% RSLogix 500 project SARUUU_BAK000.RSS, saved by version 8.10.00.18 %
PROJECT "UNTITLED"    % processor: MicroLogix 1200 %

PROGRAM FILES
  LAD 2   3 rungs

DATA FILES
  O0 OUTPUT  4 elements
  I1 INPUT  4 elements
  S2 STATUS  66 elements
  B3 BINARY  1 elements
  T4 TIMER  1 elements
  C5 COUNTER  1 elements
  R6 CONTROL  1 elements
  N7 INTEGER  1 elements

LADDER 2
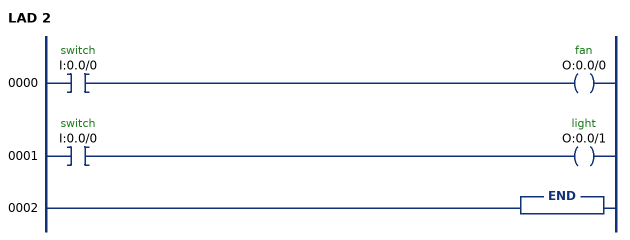
% Rung: 0 %  % edit flag set %
SOR XIC I:0.0/0 OTE O:0.0/0 EOR
%   I:0.0/0  "switch" %
%   O:0.0/0  "fan" %
% Rung: 1 %  % edit flag set %
SOR XIC I:0.0/0 OTE O:0.0/1 EOR
%   I:0.0/0  "switch" %
%   O:0.0/1  "light" %
% Rung: 2 %
SOR END EOR
